Fanuc KAREL source: kt00536.KL

-- PROVISIONAL review KL for V1013-1; original PC SHA256 ed39c0d8ecf213d1c5fd4b2aa3a86a887f8a8a33be48c33490500b086bd850d8
-- Incomplete behavior may be omitted. Consult companion uncertainty JSON. Do not deploy.
PROGRAM KT00536
%NOLOCKGROUP
-- UNRESOLVED_DECL P1 type=000199
-- UNRESOLVED_DECL P2 type=000101
-- UNRESOLVED_DECL OUT type=000106
BEGIN
  -- UNRESOLVED_PC offsets 5-39; opcodes 49,7E,49,60,7E,4A
  -- UNRESOLVED_PC offsets 44-48; opcodes 7F
END KT00536
